// TIA Portal V20 export
TYPE "typeCmControlNodeSoftCamjrUnIoadingPnPAxisX"
// stored: Namespace Unit1.Em13
   STRUCT
      pos00_wait : "LER_typeSoftCamPosition";
      pos01_workReady : "LER_typeSoftCamPosition";
      pos02_weightCheck : "LER_typeSoftCamPosition";
      pos03_conveyorQrRead : "LER_typeSoftCamPosition";
      pos04_conveyorLoad : "LER_typeSoftCamPosition";
      pos05_stackNgBox : "LER_typeSoftCamPosition";
      pos06_posistion : "LER_typeSoftCamPosition";
      pos07_posistion : "LER_typeSoftCamPosition";
      pos08_posistion : "LER_typeSoftCamPosition";
      pos09_posistion : "LER_typeSoftCamPosition";
      pos10_posistion : "LER_typeSoftCamPosition";
      pos11_posistion : "LER_typeSoftCamPosition";
      pos12_posistion : "LER_typeSoftCamPosition";
      pos13_posistion : "LER_typeSoftCamPosition";
      pos14_posistion : "LER_typeSoftCamPosition";
      pos15_posistion : "LER_typeSoftCamPosition";
   END_STRUCT;
END_TYPE
